{attribute 'enable_dynamic_creation'}
FUNCTION_BLOCK FB_ROS2Camera EXTENDS FB_Camera
VAR
	// ROS2 Camera specific properties
END_VAR

// ROS2 Camera implementation

END_FUNCTION_BLOCK

(* stored: Version 1.1.0.1
   POU FB_ROS2Camera: Id {f1b2c3d4-5557-5555-5555-555555555555} *)
